KUKA KRL program: PEGINHOLE2.src, PEGINHOLE2.dat

--- PEGINHOLE2.src ---
&ACCESS RVP
&REL 21
&PARAM TEMPLATE = C:\KRC\Roboter\Template\vorgabe
&PARAM EDITMASK = *
DEF PEGINHOLE2( )
DECL FRAME PT1
DECL BOOL TEMP
DECL BOOL STATE

DECL IPO_MODE LAST_IPO
;FOLD INI
  ;FOLD BASISTECH INI
    GLOBAL INTERRUPT DECL 3 WHEN $STOPMESS==TRUE DO IR_STOPM ( )
    INTERRUPT ON 3
    BAS (#INITMOV,0 )
  ;ENDFOLD (BASISTECH INI)
  ;FOLD USER INI
    ;Make your modifications here

  ;ENDFOLD (USER INI)
;ENDFOLD (INI)

$TOOL=TOOL_DATA[5]
$VEL.CP=.2
$VEL.ORI1=100
$VEL.ORI2=100
$ACC.CP=1.0
$ACC.ORI1=80
$ACC.ORI2=80
$ADVANCE=5

;FOLD PTP P0 Vel=100 % PDAT0 Tool[5]:Pneumatic_gripper_probe Base[0];%{PE}%R 5.6.11,%MKUKATPBASIS,%CMOVE,%VPTP,%P 1:PTP, 2:P0, 3:, 5:100, 7:PDAT0
$BWDSTART=FALSE
PDAT_ACT=PPDAT0
FDAT_ACT=FP0
BAS(#PTP_PARAMS,100)
PTP XP0
;ENDFOLD


;PT1=GETPOINT("Z", -1)
;PTP PT1

;LIN_REL{X -40}


TEMP=TRIG()
TEMP=SETSTIFF("Z", 10.0)

LIN_REL{Z -12}

STATE = STARTIMPEDANCE(TRUE)

WAIT SEC 2

LAST_IPO = $IPO_MODE
$IPO_MODE = #TCP

; Clear all search parameters
STATE = CANCEL_SEARCH()

STATE = STATE AND ADDTERMCLOCK(#ALARMCLOCK, #FAIL, 40000.0, 5)
STATE = STATE AND ADDTERMDISTANCE(#SUCCESS, 0.0, 0.0, 12.0, 0.0)

; Spiral Test

;BOOL ADDSEARCHSPIRAL(INT TURNS, REAL RADIUS, REAL SPEED)
STATE = ADDSEARCHSPIRAL(10, 30.0, 50.0)
STATE = STATE AND ADDSEARCHLINEAR(0.0, 0.0, -40.0, 10.0)

WHILE STATE
  STATE = (SEARCH() == #RUNNING)
ENDWHILE

WAIT SEC 2
LIN_REL{Z 200}

TEMP=FORCEZSTOP()
$STIFFNESS.STRATEGY=10
$STIFFNESS.COMMIT=TRUE

STATE=STARTIMPEDANCE(FALSE)

STATE = CANCEL_SEARCH()
WAIT SEC 2


;FOLD PTP P1 Vel=100 % PDAT1 Tool[5]:Pneumatic_gripper_probe Base[0];%{PE}%R 5.6.11,%MKUKATPBASIS,%CMOVE,%VPTP,%P 1:PTP, 2:P1, 3:, 5:100, 7:PDAT1
$BWDSTART=FALSE
PDAT_ACT=PPDAT1
FDAT_ACT=FP1
BAS(#PTP_PARAMS,100)
PTP XP1
;ENDFOLD


END

--- PEGINHOLE2.dat ---
&ACCESS RVP
&REL 21
&PARAM TEMPLATE = C:\KRC\Roboter\Template\vorgabe
&PARAM EDITMASK = *
DEFDAT  PEGINHOLE2
;FOLD EXTERNAL DECLARATIONS;%{PE}%MKUKATPBASIS,%CEXT,%VCOMMON,%P
;FOLD BASISTECH EXT;%{PE}%MKUKATPBASIS,%CEXT,%VEXT,%P
EXT  BAS (BAS_COMMAND  :IN,REAL  :IN )
DECL INT SUCCESS
;ENDFOLD (BASISTECH EXT)
;FOLD USER EXT;%{E}%MKUKATPUSER,%CEXT,%VEXT,%P
;Make here your modifications

;ENDFOLD (USER EXT)
;ENDFOLD (EXTERNAL DECLARATIONS)
DECL BASIS_SUGG_T LAST_BASIS={POINT1[] "P1                      ",POINT2[] "P1                      ",CP_PARAMS[] "CPDAT0                  ",PTP_PARAMS[] "PDAT1                   ",CONT[] "                        ",CP_VEL[] "2.0                     ",PTP_VEL[] "100                     ",SYNC_PARAMS[] "SYNCDAT                 ",SPL_NAME[] "S0                      "}
DECL PDAT PPDAT0={VEL 100.0,ACC 100.0,APO_DIST 100.0,APO_MODE #CPTP}
DECL E6POS XP0={X -385.334015,Y -522.388672,Z 11.8551903,A 10.2247801,B -0.0956432074,C 179.211395,S 1,T 44,E1 1.45407498,E2 0.0,E3 0.0,E4 0.0,E5 0.0,E6 0.0}
DECL FDAT FP0={TOOL_NO 5,BASE_NO 0,IPO_FRAME #BASE,POINT2[] " ",TQ_STATE FALSE}
DECL E6POS XP1={X -103.313499,Y -581.921997,Z 236.496399,A 8.40300846,B -1.84802997,C 173.704102,S 1,T 36,E1 2.22721195,E2 0.0,E3 0.0,E4 0.0,E5 0.0,E6 0.0}
DECL FDAT FP1={TOOL_NO 5,BASE_NO 0,IPO_FRAME #BASE,POINT2[] " ",TQ_STATE FALSE}
DECL PDAT PPDAT1={VEL 100.0,ACC 100.0,APO_DIST 100.0,APO_MODE #CPTP}
DECL E6POS XP2={X -284.647003,Y -616.365295,Z -15.4491501,A -23.6703091,B 1.04149604,C 179.662094,S 1,T 44,E1 -0.0126686096,E2 0.0,E3 0.0,E4 0.0,E5 0.0,E6 0.0}
DECL FDAT FP2={TOOL_NO 5,BASE_NO 0,IPO_FRAME #BASE,POINT2[] " ",TQ_STATE FALSE}
DECL PDAT PPDAT2={VEL 100.0,ACC 100.0,APO_DIST 100.0,APO_MODE #CPTP}
ENDDAT
